Yaskawa INFORM job: TEST_SCAN_FOTO_LINEAR.JBI

/JOB
//NAME TEST_SCAN_FOTO_LINEAR
///FOLDERNAME TEST_JOBS
//POS
///NPOS 0,0,0,1,0,0
///USER 4
///TOOL 1
///POSTYPE USER
///RECTAN
///RCONF 1,0,0,0,0,0,0,0,0,0,0,0,0,0,0,0,0,0,0,0,0,0,0,0
P00100=-51.450,-41.710,12.601,0.0000,0.0000,0.0000
//ALIAS
///LVARS 0,0,2,0,0,2,0,0
LD000 USERFRAME
LD001 V_SCAN
LP000 PKT_1
LP001 PKT_2
//INST
///DATE 2022/11/08 16:22
///ATTR SC,RW
///GROUP1 RB1
///LVARS 0,0,2,0,0,2,0,0
NOP
CALL JOB:TRIGGER_RESET
SET USERFRAME 4
'SCAN-GESCHWINDIGKEIT
'       [mm/s]
CALL JOB:GET_V ARGF20 ARGF"mm/s"
GETS V_SCAN $RV
'USERFRAME IN TC SETZEN
CALL JOB:SET_UFRAME ARGFUSERFRAME
'PUNKTE ERZEUGEN
CALL JOB:PUNKTE_ERZEUGEN_UF ARGFUSERFRAME ARGF100000 ARGF90000 ARGF0
SET PKT_1 P100
CALL JOB:PUNKTE_ERZEUGEN_UF ARGFUSERFRAME ARGF200000 ARGF90000 ARGF0
SET PKT_2 P100
CALL JOB:TRIGGER ARGF"PROGRAMM_EIN"
CALL JOB:SCAN_LINEAR_ARG_P ARGFPKT_1 ARGFPKT_2 ARGF15000 ARGFV_SCAN
CALL JOB:TAKE_PICTURES_OF_LINEAR_TRACE ARGFPKT_2 ARGFPKT_1 ARGFUSERFRAME ARGF40000
CALL JOB:TRIGGER ARGF"PROGRAMM_AUS"
CALL JOB:TRIGGER_RESET
END
